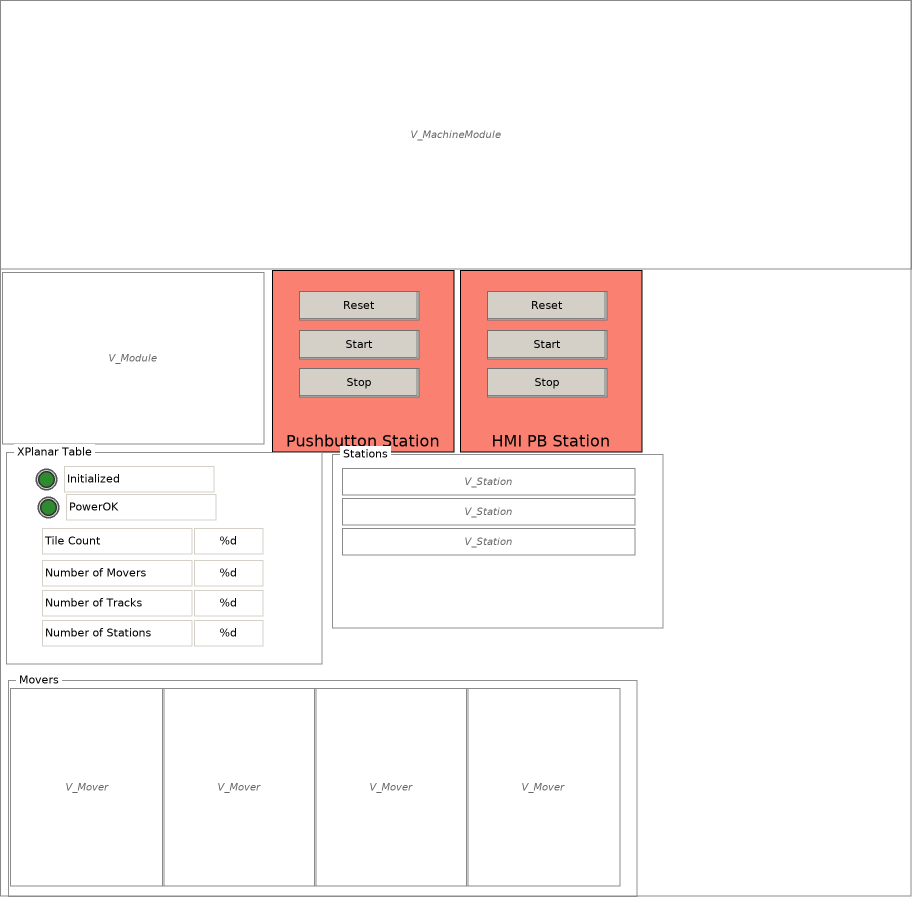
VISUALIZATION V_Main  // 912x897
    GroupBox (8,672 629x225), "Movers"
        Frame (2,16 154x198)
            shows V_Mover(Mover := MAIN.Machine.XPlanar.XPlanarTable._Movers[1].Mover_HMI, Position := MAIN.Machine.XPlanar.XPlanarTable._Movers[1]._Mover.ActPos)
        Frame (154,16 154x198)
            shows V_Mover(Mover := MAIN.Machine.XPlanar.XPlanarTable._Movers[2].Mover_HMI, Position := MAIN.Machine.XPlanar.XPlanarTable._Movers[2]._Mover.ActPos)
        Frame (306,16 154x198)
            shows V_Mover(Mover := MAIN.Machine.XPlanar.XPlanarTable._Movers[3].Mover_HMI, Position := MAIN.Machine.XPlanar.XPlanarTable._Movers[3]._Mover.ActPos)
        Frame (458,16 154x198)
            shows V_Mover(Mover := MAIN.Machine.XPlanar.XPlanarTable._Movers[4].Mover_HMI, Position := MAIN.Machine.XPlanar.XPlanarTable._Movers[4]._Mover.ActPos)
    Frame (0,0 912x269)
        shows V_MachineModule(HMI := MAIN.Machine.PackMLBaseModule_HMI)
    Frame (2,272 262x172)
        shows V_Module(HMI := MAIN.Machine.XPlanar.PackMLBaseModule_HMI)
    Group (272,270 182x175)
        RoundedRectangle (0,0 182x182), "Pushbutton Station"
        Button (27,98 120x29), "Stop", input disabled if: not MAIN.ControlSourcePB.MainPMLControl_Simplified.StopPermissive
            tap MAIN.ControlSourcePB.MainPMLControl_Simplified.StopPressed
        Button (27,21 120x29), "Reset", input disabled if: not MAIN.ControlSourcePB.MainPMLControl_Simplified.ResetPermissive
            tap MAIN.ControlSourcePB.MainPMLControl_Simplified.ResetPressed
        Button (27,60 120x29), "Start", input disabled if: not MAIN.ControlSourcePB.MainPMLControl_Simplified.StartPermissive
            tap MAIN.ControlSourcePB.MainPMLControl_Simplified.StartPressed
    Group (460,270 182x175)
        RoundedRectangle (0,0 182x182), "HMI PB Station"
        Button (27,98 120x29), "Stop", input disabled if: not MAIN.ControlSourceHMI.MainPMLControl_Simplified.StopPermissive
            tap MAIN.ControlSourceHMI.MainPMLControl_Simplified.StopPressed
        Button (27,21 120x29), "Reset", input disabled if: not MAIN.ControlSourceHMI.MainPMLControl_Simplified.ResetPermissive
            tap MAIN.ControlSourceHMI.MainPMLControl_Simplified.ResetPressed
        Button (27,60 120x29), "Start", input disabled if: not MAIN.ControlSourceHMI.MainPMLControl_Simplified.StartPermissive
            tap MAIN.ControlSourceHMI.MainPMLControl_Simplified.StartPressed
    Group (332,446 331x219)
        Frame (10,22 293x27)
            shows V_Station(Station := MAIN.Machine.XPlanar.Station1.Station_HMI)
        Frame (10,52 293x27)
            shows V_Station(Station := MAIN.Machine.XPlanar.Station2.Station_HMI)
        Frame (10,82 293x27)
            shows V_Station(Station := MAIN.Machine.XPlanar.Station3.Station_HMI)
        GroupBox (0,0 331x182), "Stations"
    Group (6,444 316x220)
        Lamp1 (28,23 25x25), variable: MAIN.Machine.XPlanar.XPlanarTable.XPlanar_HMI.Status.Initialized, style: Lamp-Lamp1-Green
        Textfield (58,22 150x26), "Initialized"
        Lamp1 (30,51 25x25), variable: MAIN.Machine.XPlanar.XPlanarTable.XPlanar_HMI.Status.PowerOK, style: Lamp-Lamp1-Green
        Textfield (60,50 150x26), "PowerOK"
        Textfield (188,84 69x26), "%d", text variable: MAIN.Machine.XPlanar.XPlanarTable.XPlanar_HMI.Status.TileCount
        Textfield (36,84 150x26), "Tile Count"
        Textfield (188,116 69x26), "%d", text variable: MAIN.Machine.XPlanar.XPlanarTable.XPlanar_HMI.Status.NumberOfMovers
        Textfield (36,116 150x26), "Number of Movers"
        Textfield (188,146 69x26), "%d", text variable: MAIN.Machine.XPlanar.XPlanarTable.XPlanar_HMI.Status.NumberOfTracks
        Textfield (36,146 150x26), "Number of Tracks"
        Textfield (188,176 69x26), "%d", text variable: MAIN.Machine.XPlanar.XPlanarTable.XPlanar_HMI.Status.NumberOfStations
        Textfield (36,176 150x26), "Number of Stations"
        GroupBox (0,0 316x220), "XPlanar Table"
END_VISUALIZATION

(* stored: Version 1.1.0.1, ProductVersion 3.1.4024.12
   Visu V_Main: Id {a820fc1e-d71f-479f-a200-f2cc0d18dc0b} *)
